{attribute 'GeneratedUsingTerminal: EK1100-0000-0018'}
{attribute addProperty BoxType "EK1100-0000-0018"}
{attribute addProperty Id "Beckhoff_EPP4xxxEK1122Beckhoff_EPP4xxxEK1122_7B2A71B7166"}
{attribute addProperty CRC "4184281145"}
{attribute addProperty Size "166"}
TYPE Beckhoff_EPP4xxx_F9671039 EXTENDS EK1100_1FC0878B :
STRUCT
	{attribute addProperty Name "Beckhoff_EPP4xxxEK1122"}
	{attribute addProperty PreviousPort "Beckhoff EPP4xxx : B"}
	Beckhoff_EPP4xxxEK1122 : Beckhoff_EPP4xxxEK1122_7B2A71B7;
END_STRUCT
END_TYPE

(* stored: Version 1.2.0.0, ProductVersion 3.1.4024.9
   DUT Beckhoff_EPP4xxx_F9671039: Id {47384451-c6d6-4650-9004-82cd3d4ba33d} *)
